{attribute 'qualified_only'}
{attribute 'strict'}
{attribute 'to_string'}
TYPE E_SelectorSwitchPos :
(
	Up := 0,
	Left:=1,
	Right:=2
)BYTE;
END_TYPE

(* stored: Version 1.1.0.1, ProductVersion 3.1.4026.19
   DUT E_SelectorSwitchPos: Id {12881b3e-30fb-4b3b-8275-4cf8018f5f1a} *)
